FUNCTION_BLOCK FB_LamparaAsignada_IL
// La lampara se enciende mientras se acciona el pulsador
VAR
    Lampara AT %Q*: BOOL;
    Pulsador AT %I*: BOOL;
END_VAR

// NETWORK 1
// instruction list
LD      Pulsador
ST      Lampara

END_FUNCTION_BLOCK

(* stored: Version 1.1.0.1, ProductVersion 3.1.4024.15
   POU FB_LamparaAsignada_IL: Id {e8f500ad-30a5-421a-8fe0-540626e93b60}, SpecialFunc None *)
